Staubli VAL3: init.pgx

public program init()
begin

  // Initialize UI

  userPage("uxMonitor")

end
